// TIA Portal V20 export
VAR_GLOBAL   // PLC tag table "BarcodeReader_DP4"
   "DP4-TriggerEnable" AT %Q294.0 : Bool;
   "DP4-Trigger" AT %Q294.1 : Bool;
   "DP4-TriggerReady" AT %I318.0 : Bool;
   "DP4-TriggerAck" AT %I318.1 : Bool;
   "DP4-Acquiring" AT %I318.2 : Bool;
   "DP4-MissedAcq" AT %I318.3 : Bool;
   "DP4-TriggerID" AT %IW319 : Word;
   "DP4-BufferResultsEnable" AT %Q295.0 : Bool;
   "DP4-ResultsAck" AT %Q295.1 : Bool;
   "DP4-Decoding" AT %I321.0 : Bool;
   "DP4-Decode Complete" AT %I321.1 : Bool;
   "DP4-Results Buffer Overrun" AT %I321.2 : Bool;
   "DP4-Results Available" AT %I321.3 : Bool;
   "DP4-General Fault" AT %I321.7 : Bool;
   "DP4-Train Code" AT %Q296.0 : Bool;
   "DP4-Train Match String" AT %Q296.1 : Bool;
   "DP4-Train Focus" AT %Q296.2 : Bool;
   "DP4-Train Brightness" AT %Q296.3 : Bool;
   "DP4-Untrain" AT %Q296.4 : Bool;
   "DP4-Execute DMCC" AT %Q296.6 : Bool;
   "DP4-Set Match String" AT %Q296.7 : Bool;
   "DP4-Train Code Ack" AT %I322.0 : Bool;
   "DP4-Train Match String Ack" AT %I322.1 : Bool;
   "DP4-Train Focus Ack" AT %I322.2 : Bool;
   "DP4-Train Brightness Ack" AT %I322.3 : Bool;
   "DP4-Untrain Ack" AT %I322.4 : Bool;
   "DP4-Execute DMCC Ack" AT %I322.6 : Bool;
   "DP4-Set Match String Ack" AT %I322.7 : Bool;
   "DP4-UserData Option" AT %QW297 : Word;
   "DP4-UserData Length" AT %QW299 : Word;
   "DP4-UserData[0]" AT %QB301 : Byte;
   "DP4-UserData[1]" AT %QB302 : Byte;
   "DP4-UserData[2]" AT %QB303 : Byte;
   "DP4-UserData[7]" AT %QB308 : Byte;
   "DP4-UserData[8]" AT %QB309 : Byte;
   "DP4-UserData[14]" AT %QB315 : Byte;
   "DP4-UserData[15]" AT %QB316 : Byte;
   "DP4-ResultID" AT %IW323 : Word;
   "DP4-Result Code" AT %IW326 : Word;
   "DP4-Read / No Read" AT %I326.0 : Bool;
   "DP4-Validated / Not Validated" AT %I326.1 : Bool;
   "DP4-Verified / Not Verified" AT %I326.2 : Bool;
   "DP4-Acquisition Trigger Overrun" AT %I326.3 : Bool;
   "DP4-Acquisition Buffer Overflow" AT %I326.4 : Bool;
   "DP4-Result Extended" AT %IW327 : Word;
   "DP4-InspectionResults[10]" AT %IB341 : Byte;
   "DP4-InspectionResults[11]" AT %IB342 : Byte;
   "DP4-InspectionResults[12]" AT %IB343 : Byte;
   "DP4-InspectionResults[13]" AT %IB344 : Byte;
   "DP4-InspectionResults[14]" AT %IB345 : Byte;
   "DP4-InspectionResults[15]" AT %IB346 : Byte;
   ContinousGetResults_DP4 AT %M10.1 : Bool;
   TrainFocus_DP4 AT %M10.2 : Bool;
   "DP4-Result Length" AT %IW329 : Word;
   "DP4-InspectionResults[0]" AT %IB331 : Byte;
   "DP4-InspectionResults[1]" AT %IB332 : Byte;
   "DP4-InspectionResults[2]" AT %IB333 : Byte;
   "DP4-InspectionResults[3]" AT %IB334 : Byte;
   "DP4-InspectionResults[4]" AT %IB335 : Byte;
   "DP4-InspectionResults[5]" AT %IB336 : Byte;
   "DP4-InspectionResults[6]" AT %IB337 : Byte;
   "DP4-InspectionResults[7]" AT %IB338 : Byte;
   "DP4-InspectionResults[8]" AT %IB339 : Byte;
   "DP4-InspectionResults[9]" AT %IB340 : Byte;
   "Result data_DP4" AT %I331.0 : "Global.BarCode";
   "DP4-UserData[3]" AT %QB304 : Byte;
   "DP4-UserData[4]" AT %QB305 : Byte;
   "DP4-UserData[5]" AT %QB306 : Byte;
   "DP4-UserData[6]" AT %QB307 : Byte;
   "DP4-UserData[9]" AT %QB310 : Byte;
   "DP4-UserData[10]" AT %QB311 : Byte;
   "DP4-UserData[11]" AT %QB312 : Byte;
   "DP4-UserData[12]" AT %QB313 : Byte;
   "DP4-UserData[13]" AT %QB314 : Byte;
   UserData_DP4 AT %Q301.0 : "Global.BarCode";
END_VAR
